// TIA Portal V20 export
// export: Created 2025-12-01T14:57:19.9583776Z, ExportSetting None, DisplayName Totally Integrated Automation Portal, DisplayVersion V20 Update 3, DisplayName TIA Portal Openness, DisplayVersion V20 Update 3, DisplayName TIA Portal Version Control Interface, DisplayVersion V20 Update 3, DisplayName STEP 7 Professional, DisplayVersion V20 Update 3, DisplayName STEP 7 Safety, DisplayVersion V20 Update 2, DisplayName WinCC Basic/Comfort/Advanced, DisplayVersion V20 Update 3, DisplayName WinCC Professional, DisplayVersion V20 Update 3, DisplayName WinCC Unified, DisplayVersion V20 Update 3
DATA_BLOCK "DB940_Datos_VAR_Lenze_i550"   // DB940
{ S7_Optimized_Access := 'FALSE' }
// stored: AutoNumber false
   VAR RETAIN
      Lenze_i550 : Array[0..255] of Struct
         "Estatus variador" { S7_SetPoint := 'True'} : "i550 Estatus variador";   // Word que informa del estado del dispositivo
         "Código de error" : UInt;   // Código proporcionado por Lenze para diagnosticar el fallo
         "Frecuencia actual" : Int;   // Frecuencia actual en dispositivo. Formato 3250 = 32,50 Hz
         "Corriente actual" : Int;   // Corriente actual en dispositivo. Formato 21 = 2,1 A
         "Posicion encoder" : Real;   // Posición actual (solo con encoder) Formato Inc x vuelta motor
         "Palabra de control" { S7_SetPoint := 'True'} : "i550 Palabra de control";   // Word que controla la activación del dispositvo
         "Consigna de frecuencia" : Int;   // Frecuencia enviada al dispositivo. Formato 3250 = 32,50 Hz
         ACC : Int;   // 5->0,5sg; 10->1sg; 50->5sg; 100->10sg a Frecuencia máxima
         DCC : Int;   // 5->0,5sg; 10->1sg; 50->5sg; 100->10sg a Frecuencia máxima
         Termico_Tx : Bool;
      END_STRUCT;
   END_VAR
BEGIN
   Lenze_i550[0..2].ACC := 50;
   Lenze_i550[3].ACC := 10;
   Lenze_i550[4..41].ACC := 50;
   Lenze_i550[42..43].ACC := 10;
   Lenze_i550[44..199].ACC := 50;
   Lenze_i550[200].ACC := 10;
   Lenze_i550[201..255].ACC := 50;
   Lenze_i550[0..2].DCC := 50;
   Lenze_i550[3].DCC := 10;
   Lenze_i550[4..41].DCC := 50;
   Lenze_i550[42..43].DCC := 10;
   Lenze_i550[44..199].DCC := 50;
   Lenze_i550[200].DCC := 10;
   Lenze_i550[201..255].DCC := 50;
END_DATA_BLOCK
